Universal Robots PolyScope program: test.urp

Program test (installation=default directory=/root/ursim/programs createdIn=5.11.11.1010533 lastSavedIn=5.11.11.1010533 robotSerialNumber=20195599999)
Calibrated DH parameters: a=[0, -0.425, -0.3922, 0, 0, 0]; d=[0.1625, 0, 0, 0.1333, 0.0997, 0.0996]; alpha=[1.570796, 0, 0, 1.570796, -1.570796, 0]; deltaTheta=[0, 0, 0, 0, 0, 0]
Robot Program (runOnlyOnce=false)
  Placeholder
